Universal Robots URScript: 00C_03_JieXian_BiRang.script

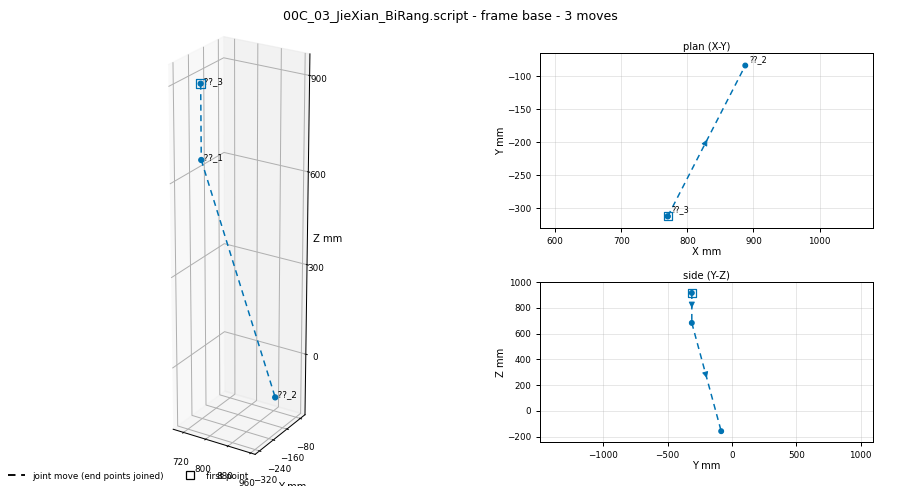
[picture p0: tool path of 00C_03_JieXian_BiRang.script in frame base, 3 of 3 moves have a stored position in this frame; points joined in program order, loops and branches not executed]
def P00C_03_JieXian_BiRang():
  set_gravity([0.0, 0.0, 9.82])
  set_safety_mode_transition_hardness(1)
  set_standard_analog_input_domain(0, 1)
  set_standard_analog_input_domain(1, 1)
  set_tool_analog_input_domain(0, 1)
  set_tool_analog_input_domain(1, 1)
  set_analog_outputdomain(0, 0)
  set_analog_outputdomain(1, 0)
  set_tool_voltage(24)
  set_input_actions_to_default()
  set_tcp(p[0.0,0.0,0.32,0.0,0.0,-0.5236])
  set_payload(8.0)
  global Zhua_1=[0.08063, -2.42649, -1.72682, -0.47876, 0.40808, -1.10831]
  global prepose=p[0.98979, -0.16931, -0.39963, 1.98720, 0.07234, 0.05469]
  global i_var_2=0
  global i_var_1=True
  global pose=p[0.98979, -0.31931, -0.39963, 1.98720, 0.07234, 0.05469]
  $ 1 "机器人程序"
  $ 2 "MoveJ"
  $ 3 "路点_3"
  set_tcp(p[-0.06262,0.03599,0.32923,0.0,0.0,1.3731])
  movej(get_inverse_kin(p[.770210656907, -.311925180187, .915354097022, .061495088104, -.011895324032, 1.533264379946], qnear=[-0.18626290956606084, -1.9358022848712366, -1.5686381498919886, -1.2483838240252894, -1.5420282522784632, -1.2265570799456995]), a=0.6981317007977318, v=0.5235987755982988)
  $ 4 "路点_1"
  set_tcp(p[-0.06262,0.03599,0.32923,0.0,0.0,1.3731])
  movej(get_inverse_kin(p[.770282550510, -.311966737125, .682450112893, .061618605549, -.012162098221, 1.533427942792], qnear=[-0.18573552766908819, -2.13527757326235, -1.7365315596209925, -0.8810747305499476, -1.5408299604998987, -1.2232630888568323]), a=0.6981317007977318, v=0.5235987755982988)
  $ 5 "路点_2"
  set_tcp(p[-0.06262,0.03599,0.32923,0.0,0.0,1.3731])
  movej(get_inverse_kin(p[.887554999183, -.083733032097, -.158806531755, .567007366793, .631363737733, 1.439451240319], qnear=[0.06396542489528656, -3.117643181477682, -1.7016404310809534, -0.6665790716754358, -1.5575783888446253, -1.473001782094137]), a=0.6981317007977318, v=0.5235987755982988)
end
